Staubli VAL3: getMaxNumOfPart.pgx

public program getMaxNumOfPart(num& x_nMaxNumOfPart[])
begin
  // This program returns the size of the buffer
  // The buffer size represents the maximum number of parts
  // that can be simultaneously detected by the detection device
  x_nMaxNumOfPart=nMaxNumOfObject
end
